# EPICS substitutions: apps/jscalerApp/Db/wf/jscalers_wf_S6.substitutions
file "db/jscalers_wf_averages-1type-1sector.db" {
pattern { T S }
{ FADC 6 }
{ TRG 6 }
{ TDC 6 }
}
